PROGRAM PRG_SystemInit
VAR_OUTPUT
	bDone           : BOOL := FALSE;
END_VAR
VAR
	i               : INT;
	j				: INT;
    bAllDone        : BOOL := FALSE;
    bStartedAction  : BOOL := FALSE;
	bMoveZeroDone	: BOOL := FALSE;
    bInitComplete   : BOOL := FALSE;
	bVerticalMotorsDone		: BOOL := FALSE;   
	bLinearMotorsHomingDone	: BOOL := FALSE; 
	bValvesHomingDone 		: BOOL := FALSE;
	bLinearPumpsDone		: BOOL := FALSE;
	bPerformHoming			: BOOL := FALSE;
	
	bAllResetDone		: BOOL := FALSE;
	bEnableDone			: BOOL := FALSE;
	bResetCheck			: ARRAY[1..28] OF BOOL;
	
	aMotorsEnabled 	: ARRAY[1..3] OF BOOL;
	aValvesEnabled 	: ARRAY[1..5] OF BOOL;
	aLinearPumpsEnabled	: ARRAY[1..10] OF BOOL;
	aRotaryPumpsEnabled	: ARRAY[1..10] OF BOOL;
	
	bAllPumpsEnabled  : BOOL := FALSE;
	bAllLinearPumpsEnabled  : BOOL := FALSE;
	bAllRotaryPumpsEnabled  : BOOL := FALSE;
	bAllMotorsEnabled : BOOL := FALSE;
	bAllValvesEnabled : BOOL := FALSE;
	
	bHomeMotorDone	: ARRAY[1..3] OF BOOL;
	bHomeValveDone  : ARRAY[1..5] OF BOOL;
	bHomePumpDone	: ARRAY[1..10] OF BOOL;
	
	bM2InPosition	: BOOL;
	rPosTolerance	: REAL := 1.0;
	
	bMoveValve1Request	: BOOL := TRUE;
	bMoveValve2Request	: BOOL := TRUE;
	
	bMoveMotorsRequest	: ARRAY[1..3] OF BOOL;
	bMoveMotorDone		: ARRAY[1..3] OF BOOL;
	
	bCalibrationReset	  : BOOL := FALSE;
	bManualModeReset	  : BOOL := FALSE;
	bAutoCycleReset		  : BOOL := FALSE;
	bAllLogicResetDone	  : BOOL := FALSE;
	bInitLogicLatchesDone : BOOL := FALSE;
	
	tonResetDelay	: ton;
	tonEnableDelay	: ton;
	
	//Timeout timers for each step
	tonResetTimeOut		: ton;
	tonEnableTimeOut	: ton;
	tonHomeTimeOut		: ton;
	tonMoveAbsTimeOut	: ton;
		
	stStatus : ST_ActuatorStatus;
	
END_VAR

// ============================================================================
// PRG_SystemInit
// Handles full system initialization sequence:
//  0) Reset PRG's Manual | Calibration | AutoCycle
//  1) Reset all axes (motors, valves, pumps)
//  2) Enable all required axes
//  3) Perform homing on first startup OR move axes to zero on subsequent inits
//  4) Check completion and errors
//  5) Set bDone when initialization is complete
// ============================================================================

// ---------------------------------------------------------------------------
// 0) Basic delays between phases
// ---------------------------------------------------------------------------

// Delay before starting Reset
tonResetDelay(
    IN := NOT bAllResetDone,
    PT := T#1S
);

// Delay before starting Enable (only after Reset is fully done)
tonEnableDelay(
    IN := bAllResetDone AND NOT bEnableDone,
    PT := T#1S
);

// ---------------------------------------------------------------------------
// 0) Step 0 - Reset all logic Flags, PRGs and FBs
// ---------------------------------------------------------------------------
IF NOT bInitLogicLatchesDone THEN ACT_ResetCommandFlags(); END_IF

IF NOT bAllLogicResetDone AND bInitLogicLatchesDone THEN ACT_LogicResets(); END_IF

// ---------------------------------------------------------------------------
// 1) Step 1 - Reset all axes (motors, valves, linear and rotary pumps)
// ---------------------------------------------------------------------------
IF NOT bAllResetDone AND bAllLogicResetDone AND bInitLogicLatchesDone AND tonResetDelay.Q THEN
    ACT_ResetMotors();   // Uses bResetCheck[1..28], tonResetTimeOut, etc.
END_IF

// ---------------------------------------------------------------------------
// 2) Step 2 - Enable all axes (motors, valves, rotary pumps)
//     - Uses extra layer: checks Axis.Status.Error before/after Enable
// ---------------------------------------------------------------------------
IF bAllResetDone AND NOT bEnableDone AND tonEnableDelay.Q THEN
    ACT_EnableMotors();
END_IF

// ---------------------------------------------------------------------------
// 3) Step 3 - Decide if we need Homing or only MoveToZero
//     - First SystemInit: perform homing (bInitialHomingDone = FALSE)
//     - Next SystemInits: only move motors/valves to zero/home position
// ---------------------------------------------------------------------------

IF NOT bStartedAction AND bAllResetDone AND bEnableDone THEN
    bStartedAction := TRUE;

    // First time the machine starts: perform initial homing
    IF NOT GVL_Motion.bInitialHomingDone THEN
        bPerformHoming := TRUE;   // ACT_Homing() will be called
    ELSE
        bPerformHoming := FALSE;  // ACT_MoveToZero() will be called
    END_IF
END_IF

// ---------------------------------------------------------------------------
// 3a) Execute Homing or MoveToZero depending on bPerformHoming
// ---------------------------------------------------------------------------
IF bStartedAction THEN
    IF bPerformHoming THEN
        ACT_Homing();
    ELSE
        ACT_MoveToZero();
    END_IF
END_IF

// ---------------------------------------------------------------------------
// 4) Step 4 + 5 - Check if all motors and valves have completed their action
//     - Also checks for errors from wrapper (stStatus.bError)
//       and directly from Axis.Status.Error
// ---------------------------------------------------------------------------
IF bStartedAction AND bMoveZeroDone THEN
    bAllDone := TRUE;

    // Check motors M1..M3
    FOR i := 1 TO 3 DO
        stStatus := GVL_Motion.aMotors[i].GetStatus();

        // If any motor is not done yet
        IF NOT stStatus.bDone THEN
            bAllDone := FALSE;
        END_IF

        // If any motor returned an error (wrapper OR Axis), abort with immediate fault
        IF stStatus.bError THEN
            GVL_HMI.eMachineMode := E_MachineMode.IMEDIATE_FAULT;
            RETURN;
        END_IF
    END_FOR

    // Check valves V1..V5
    FOR i := 1 TO 5 DO
        stStatus := GVL_Motion.aValvesObj[i].GetStatus();

        // If any valve is not done yet
        IF NOT stStatus.bDone THEN
            bAllDone := FALSE;
        END_IF

        // If any valve returned an error (wrapper OR Axis), abort with immediate fault
        IF stStatus.bError THEN
            GVL_HMI.eMachineMode := E_MachineMode.IMEDIATE_FAULT;
            RETURN;
        END_IF
    END_FOR
END_IF

// ---------------------------------------------------------------------------
// 5) Step 6 - Finalization of System Init
//     - Set bDone only when Reset, Enable and Actions are all completed
// ---------------------------------------------------------------------------
IF bAllDone AND bAllResetDone AND bEnableDone AND NOT bInitComplete THEN
    bInitComplete := TRUE;
    bDone         := TRUE;

    // Mark that the initial homing has been successfully completed
    IF NOT GVL_Motion.bInitialHomingDone THEN
        GVL_Motion.bInitialHomingDone := TRUE;
    END_IF
END_IF

ACTION ACT_EnableMotors:
// ============================================================================
// Step 2: Enable all motors, valves and rotary pumps
//   - Uses aMotorsEnabled[1..3], aValvesEnabled[1..5], aRotaryPumpsEnabled[1..10]
//   - Sets bAllMotorsEnabled, bAllValvesEnabled, bAllRotaryPumpsEnabled
//   - Uses tonEnableTimeOut and GVL_Alarms.sMotionEnableTimeoutAxis
//   - Extra layer: checks wrapper error (GetStatus().bError) before enabling
// ============================================================================

IF NOT bEnableDone THEN

    // Assume all will be enabled, then AND with each device
    bAllMotorsEnabled      := TRUE;
    bAllValvesEnabled      := TRUE;
    bAllRotaryPumpsEnabled := TRUE;

    // -----------------------------
    // 2.1 Motors (M1..M3)
    // -----------------------------
    FOR i := 1 TO 3 DO
        // Read wrapper status
        stStatus := GVL_Motion.aMotors[i].GetStatus();

        // If wrapper reports error at this stage, abort System Init
        IF stStatus.bError THEN
            GVL_HMI.eMachineMode := E_MachineMode.IMEDIATE_FAULT;
            RETURN;
        END_IF

        // If axis is disabled, request Enable through wrapper
        // (If your wrapper has a specific bEnabled flag, you can check it here.
        // Otherwise, just call Enable() and rely on the wrapper to handle it.)
        aMotorsEnabled[i] := GVL_Motion.aMotors[i].Enable();

        bAllMotorsEnabled := bAllMotorsEnabled AND aMotorsEnabled[i];
    END_FOR

    // -----------------------------
    // 2.2 Valves (V1..V5)
    // -----------------------------
    FOR i := 1 TO 5 DO
        stStatus := GVL_Motion.aValvesObj[i].GetStatus();

        IF stStatus.bError THEN
            GVL_HMI.eMachineMode := E_MachineMode.IMEDIATE_FAULT;
            RETURN;
        END_IF

        aValvesEnabled[i] := GVL_Motion.aValvesObj[i].Enable();

        bAllValvesEnabled := bAllValvesEnabled AND aValvesEnabled[i];
    END_FOR

    // -----------------------------
    // 2.3 Rotary pumps (RP1..RP10)
// -----------------------------
    FOR i := 1 TO 10 DO
        stStatus := GVL_Motion.aPumpsRotary[i].GetStatus();

        IF stStatus.bError THEN
            GVL_HMI.eMachineMode := E_MachineMode.IMEDIATE_FAULT;
            RETURN;
        END_IF

        aRotaryPumpsEnabled[i] := GVL_Motion.aPumpsRotary[i].Enable();

        bAllRotaryPumpsEnabled := bAllRotaryPumpsEnabled AND aRotaryPumpsEnabled[i];
    END_FOR

    // -----------------------------
    // 2.4 Enable timeout monitoring and alarm
    // -----------------------------
    tonEnableTimeOut(IN := TRUE, PT := T#10S);

    IF tonEnableTimeOut.Q AND NOT (bAllMotorsEnabled AND bAllValvesEnabled AND bAllRotaryPumpsEnabled) THEN
        // Build string with axes that were NOT enabled within timeout

        // Motors M1..M3
        FOR i := 1 TO 3 DO
            IF NOT aMotorsEnabled[i] THEN
                IF GVL_Alarms.sMotionEnableTimeoutAxis <> '' THEN
                    GVL_Alarms.sMotionEnableTimeoutAxis :=
                        CONCAT(GVL_Alarms.sMotionEnableTimeoutAxis, ', ');
                END_IF
                GVL_Alarms.sMotionEnableTimeoutAxis :=
                    CONCAT(GVL_Alarms.sMotionEnableTimeoutAxis,
                           GVL_Constant.sMotionText[i]);
            END_IF
        END_FOR

        // Valves V1..V5
        FOR i := 1 TO 5 DO
            IF NOT aValvesEnabled[i] THEN
                IF GVL_Alarms.sMotionEnableTimeoutAxis <> '' THEN
                    GVL_Alarms.sMotionEnableTimeoutAxis :=
                        CONCAT(GVL_Alarms.sMotionEnableTimeoutAxis, ', ');
                END_IF
                GVL_Alarms.sMotionEnableTimeoutAxis :=
                    CONCAT(GVL_Alarms.sMotionEnableTimeoutAxis,
                           GVL_Constant.sMotionText[i + 3]);
            END_IF
        END_FOR

        // Rotary pumps RP1..RP10
        FOR i := 1 TO 10 DO
            IF NOT aRotaryPumpsEnabled[i] THEN
                IF GVL_Alarms.sMotionEnableTimeoutAxis <> '' THEN
                    GVL_Alarms.sMotionEnableTimeoutAxis :=
                        CONCAT(GVL_Alarms.sMotionEnableTimeoutAxis, ', ');
                END_IF
                GVL_Alarms.sMotionEnableTimeoutAxis :=
                    CONCAT(GVL_Alarms.sMotionEnableTimeoutAxis,
                           GVL_Constant.sMotionText[i + 18]);
            END_IF
        END_FOR

        GVL_Alarms.bMotionEnableTimeout := TRUE;
        // Strong robustness: abort System Init on enable timeout
        GVL_HMI.eMachineMode := E_MachineMode.IMEDIATE_FAULT;
        RETURN;
    END_IF

    // -----------------------------
    // 2.5 Step completion
    // -----------------------------
    IF bAllMotorsEnabled AND bAllValvesEnabled AND bAllRotaryPumpsEnabled THEN
        bEnableDone := TRUE;
        tonEnableTimeOut(IN := FALSE);
    END_IF

ELSE
    // Already done, ensure timer is off
    tonEnableTimeOut(IN := FALSE);
END_IF
END_ACTION

ACTION ACT_Homing:
// ============================================================================
// Step 3 (part 1): Initial homing sequence
//   - Only used when GVL_Motion.bInitialHomingDone = FALSE
//   - Homes vertical motors, then horizontal motor
//   - Moves valves to home position (position 5) when positions are recovered
//   - Monitors homing timeout and raises alarm
// ============================================================================

IF bPerformHoming THEN

    // -----------------------------
    // 3.1 Vertical motors homing (M1, M2)
    // -----------------------------
    IF NOT bHomeMotorDone[1] THEN
        bHomeMotorDone[1] := GVL_Motion.aMotors[1].Home(
            pHomeSensor := ADR(GVL_IO.gDigInputs.bStageCollection_Home),
            rVelocity   := GVL_Motion.M1Motor.rHomeVel,
            rAcc        := GVL_Motion.M1Motor.rHomeAcc,
            rDec        := GVL_Motion.M1Motor.rHomeDec
        );
    END_IF

    IF NOT bHomeMotorDone[2] THEN
        bHomeMotorDone[2] := GVL_Motion.aMotors[2].Home(
            pHomeSensor := ADR(GVL_IO.gDigInputs.bSampleRecovery_Vertical_Home),
            rVelocity   := GVL_Motion.M2Motor.rHomeVel,
            rAcc        := GVL_Motion.M2Motor.rHomeAcc,
            rDec        := GVL_Motion.M2Motor.rHomeDec
        );
    END_IF

    // Check if vertical motors homing is done
    IF bHomeMotorDone[1] AND bHomeMotorDone[2] THEN
        bVerticalMotorsDone := TRUE;
    END_IF

    // -----------------------------
    // 3.2 Horizontal motor homing (M3), only after verticals are done
    // -----------------------------
    IF bVerticalMotorsDone AND NOT bHomeMotorDone[3] THEN
        bHomeMotorDone[3] := GVL_Motion.aMotors[3].Home(
            pHomeSensor := ADR(GVL_IO.gDigInputs.bSampleRecovery_Horizontal_Home),
            rVelocity   := GVL_Motion.M3Motor.rHomeVel,
            rAcc        := GVL_Motion.M3Motor.rHomeAcc,
            rDec        := GVL_Motion.M3Motor.rHomeDec
        );
    END_IF

    // Check if all linear motors are homed
    IF bHomeMotorDone[1] AND bHomeMotorDone[2] AND bHomeMotorDone[3] THEN
        bLinearMotorsHomingDone := TRUE;
    END_IF

    // -----------------------------
    // 3.3 Valves homing (move to position 5) if position is recovered
    // -----------------------------
    IF GVL_Motion.bValvesPositionRecovered THEN
        // Move all valves to position 5 (home position)
        IF NOT bHomeValveDone[1] THEN
            bHomeValveDone[1] := GVL_Motion.aValvesObj[1].MoveValve(
                iPosition := 5,
                rVelocity := GVL_Motion.aValves[1].rHomeVel,
                rAcc      := GVL_Motion.aValves[1].rHomeAcc,
                rDec      := GVL_Motion.aValves[1].rHomeDec
            );
        END_IF

        IF NOT bHomeValveDone[2] THEN
            bHomeValveDone[2] := GVL_Motion.aValvesObj[2].MoveValve(
                iPosition := 5,
                rVelocity := GVL_Motion.aValves[2].rHomeVel,
                rAcc      := GVL_Motion.aValves[2].rHomeAcc,
                rDec      := GVL_Motion.aValves[2].rHomeDec
            );
        END_IF

        IF NOT bHomeValveDone[3] THEN
            bHomeValveDone[3] := GVL_Motion.aValvesObj[3].MoveValve(
                iPosition := 5,
                rVelocity := GVL_Motion.aValves[3].rHomeVel,
                rAcc      := GVL_Motion.aValves[3].rHomeAcc,
                rDec      := GVL_Motion.aValves[3].rHomeDec
            );
        END_IF

        IF NOT bHomeValveDone[4] THEN
            bHomeValveDone[4] := GVL_Motion.aValvesObj[4].MoveValve(
                iPosition := 5,
                rVelocity := GVL_Motion.aValves[4].rHomeVel,
                rAcc      := GVL_Motion.aValves[4].rHomeAcc,
                rDec      := GVL_Motion.aValves[4].rHomeDec
            );
        END_IF

        IF NOT bHomeValveDone[5] THEN
            bHomeValveDone[5] := GVL_Motion.aValvesObj[5].MoveValve(
                iPosition := 5,
                rVelocity := GVL_Motion.aValves[5].rHomeVel,
                rAcc      := GVL_Motion.aValves[5].rHomeAcc,
                rDec      := GVL_Motion.aValves[5].rHomeDec
            );
        END_IF
    END_IF

    // Check if all valves homing are done
    bValvesHomingDone :=
        bHomeValveDone[1] AND bHomeValveDone[2] AND bHomeValveDone[3] AND
        bHomeValveDone[4] AND bHomeValveDone[5];

	// If all motors and valves completed their homing, finalize
	IF bLinearMotorsHomingDone AND bValvesHomingDone THEN 
		bMoveZeroDone := TRUE;
	END_IF	
	
    // -----------------------------
    // 3.4 Homing timeout monitoring and alarm
    // -----------------------------
    tonHomeTimeOut(
        IN := NOT (bLinearMotorsHomingDone AND bValvesHomingDone),
        PT := T#40S
    );

    IF tonHomeTimeOut.Q AND NOT (bLinearMotorsHomingDone AND bValvesHomingDone) THEN
        // Build string with axes that were NOT homed in time

        // Motors M1..M3
        FOR j := 1 TO 3 DO
            IF NOT bHomeMotorDone[j] THEN
                IF GVL_Alarms.sMotionHomeTimeoutAxis <> '' THEN
                    GVL_Alarms.sMotionHomeTimeoutAxis :=
                        CONCAT(GVL_Alarms.sMotionHomeTimeoutAxis, ', ');
                END_IF
                GVL_Alarms.sMotionHomeTimeoutAxis :=
                    CONCAT(GVL_Alarms.sMotionHomeTimeoutAxis,
                           GVL_Constant.sMotionText[j]);
            END_IF
        END_FOR

        // Valves V1..V5
        FOR j := 1 TO 5 DO
            IF NOT bHomeValveDone[j] THEN
                IF GVL_Alarms.sMotionHomeTimeoutAxis <> '' THEN
                    GVL_Alarms.sMotionHomeTimeoutAxis :=
                        CONCAT(GVL_Alarms.sMotionHomeTimeoutAxis, ', ');
                END_IF
                GVL_Alarms.sMotionHomeTimeoutAxis :=
                    CONCAT(GVL_Alarms.sMotionHomeTimeoutAxis,
                           GVL_Constant.sMotionText[j + 3]);
            END_IF
        END_FOR

        GVL_Alarms.bMotionHomeTimeout := TRUE;
        GVL_HMI.eMachineMode          := E_MachineMode.IMEDIATE_FAULT;
    END_IF

END_IF
END_ACTION

ACTION ACT_LogicResets:
IF NOT bAllLogicResetDone THEN
	
	bCalibrationReset	:= PRG_Calibration.Reset();
	bManualModeReset	:= PRG_ManualControl.Reset();
	bAutoCycleReset		:= PRG_AutoCycle.Reset();
	
	IF bCalibrationReset AND bManualModeReset AND bAutoCycleReset THEN
		bAllLogicResetDone 	:= TRUE;
	END_IF
	
END_IF
END_ACTION

ACTION ACT_MoveToZero:
// ============================================================================
// Step 3 (part 2): Move motors and valves to zero / default positions
//   - Used when GVL_Motion.bInitialHomingDone = TRUE
//   - Moves:
//       - M1, M2, M3 -> position 0.0
//       - Valves V1..V5 -> position 5
//   - Uses bMoveMotorDone[1..3] and bHomeValveDone[1..5]
//   - Monitors move absolute timeout and raises alarm
// ============================================================================

IF NOT bPerformHoming THEN

    // -----------------------------
    // 3.5 Move linear motors to 0.0
    // -----------------------------
    // You can adjust these velocity/acc/dec parameters as needed
    IF NOT bMoveMotorDone[1] THEN
        bMoveMotorDone[1] := GVL_Motion.aMotors[1].MoveAbsolute(
            rPosition := GVL_Settings.stMachineParam.aM1Position[1],
            rVelocity := GVL_Settings.stMachineParam.rM1Velocity,
            rAcc      := GVL_Settings.stMachineParam.rM1Accleration,
            rDec      := GVL_Settings.stMachineParam.rM1Deceleration
        );
    END_IF

    IF NOT bMoveMotorDone[2] THEN
        bMoveMotorDone[2] := GVL_Motion.aMotors[2].MoveAbsolute(
            rPosition := GVL_Settings.stMachineParam.aM2Position[1],
            rVelocity := GVL_Settings.stMachineParam.rM2Velocity,
            rAcc      := GVL_Settings.stMachineParam.rM2Accleration,
            rDec      := GVL_Settings.stMachineParam.rM2Deceleration
        );
    END_IF
	
	// Track real M2 Position before start moving M3 
	bM2InPosition := ABS(GVL_Motion.M2Motor.rActualPos - GVL_Settings.stMachineParam.aM2Position[1]) < rPosTolerance;
	
    IF bMoveMotorDone[2] AND bM2InPosition AND NOT bMoveMotorDone[3] THEN
        bMoveMotorDone[3] := GVL_Motion.aMotors[3].MoveAbsolute(
            rPosition := GVL_Settings.stMachineParam.aM3Position[1],
            rVelocity := GVL_Settings.stMachineParam.rM3Velocity,
            rAcc      := GVL_Settings.stMachineParam.rM3Accleration,
            rDec      := GVL_Settings.stMachineParam.rM3Deceleration
        );
    END_IF

    // Linear motors move done flag
    bLinearMotorsHomingDone :=
        bMoveMotorDone[1] AND bMoveMotorDone[2] AND bMoveMotorDone[3];

    // -----------------------------
    // 3.6 Move valves to position 5 (default/home position)
// -----------------------------
    IF NOT bHomeValveDone[1] THEN
        bHomeValveDone[1] := GVL_Motion.aValvesObj[1].MoveValve(
            iPosition := 5,
            rVelocity := GVL_Motion.aValves[1].rHomeVel,
            rAcc      := GVL_Motion.aValves[1].rHomeAcc,
            rDec      := GVL_Motion.aValves[1].rHomeDec
        );
    END_IF

    IF NOT bHomeValveDone[2] THEN
        bHomeValveDone[2] := GVL_Motion.aValvesObj[2].MoveValve(
            iPosition := 5,
            rVelocity := GVL_Motion.aValves[2].rHomeVel,
            rAcc      := GVL_Motion.aValves[2].rHomeAcc,
            rDec      := GVL_Motion.aValves[2].rHomeDec
        );
    END_IF

    IF NOT bHomeValveDone[3] THEN
        bHomeValveDone[3] := GVL_Motion.aValvesObj[3].MoveValve(
            iPosition := 5,
            rVelocity := GVL_Motion.aValves[3].rHomeVel,
            rAcc      := GVL_Motion.aValves[3].rHomeAcc,
            rDec      := GVL_Motion.aValves[3].rHomeDec
        );
    END_IF

    IF NOT bHomeValveDone[4] THEN
        bHomeValveDone[4] := GVL_Motion.aValvesObj[4].MoveValve(
            iPosition := 5,
            rVelocity := GVL_Motion.aValves[4].rHomeVel,
            rAcc      := GVL_Motion.aValves[4].rHomeAcc,
            rDec      := GVL_Motion.aValves[4].rHomeDec
        );
    END_IF

    IF NOT bHomeValveDone[5] THEN
        bHomeValveDone[5] := GVL_Motion.aValvesObj[5].MoveValve(
            iPosition := 5,
            rVelocity := GVL_Motion.aValves[5].rHomeVel,
            rAcc      := GVL_Motion.aValves[5].rHomeAcc,
            rDec      := GVL_Motion.aValves[5].rHomeDec
        );
    END_IF

    // Valves move done flag
    bValvesHomingDone :=
        bHomeValveDone[1] AND bHomeValveDone[2] AND
        bHomeValveDone[3] AND bHomeValveDone[4] AND bHomeValveDone[5];
	
	// If all motors and valves completed their homing, finalize
	IF bLinearMotorsHomingDone AND bValvesHomingDone THEN 
		bMoveZeroDone := TRUE;
	END_IF
	
    // -----------------------------
    // 3.7 MoveAbs timeout monitoring and alarm
    //    (Note: here we correctly use bMoveMotorDone instead of bHomeMotorDone)
// -----------------------------
    tonMoveAbsTimeOut(
        IN := NOT (bLinearMotorsHomingDone AND bValvesHomingDone),
        PT := T#40S
    );

    IF tonMoveAbsTimeOut.Q AND NOT (bLinearMotorsHomingDone AND bValvesHomingDone) THEN
        // Build string with axes that did NOT complete MoveAbsolute in time

        // Motors M1..M3
        FOR j := 1 TO 3 DO
            IF NOT bMoveMotorDone[j] THEN
                IF GVL_Alarms.sMotionMoveAbsTimeoutAxis <> '' THEN
                    GVL_Alarms.sMotionMoveAbsTimeoutAxis :=
                        CONCAT(GVL_Alarms.sMotionMoveAbsTimeoutAxis, ', ');
                END_IF
                GVL_Alarms.sMotionMoveAbsTimeoutAxis :=
                    CONCAT(GVL_Alarms.sMotionMoveAbsTimeoutAxis,
                           GVL_Constant.sMotionText[j]);
            END_IF
        END_FOR

        // Valves V1..V5
        FOR j := 1 TO 5 DO
            IF NOT bHomeValveDone[j] THEN
                IF GVL_Alarms.sMotionMoveAbsTimeoutAxis <> '' THEN
                    GVL_Alarms.sMotionMoveAbsTimeoutAxis :=
                        CONCAT(GVL_Alarms.sMotionMoveAbsTimeoutAxis, ', ');
                END_IF
                GVL_Alarms.sMotionMoveAbsTimeoutAxis :=
                    CONCAT(GVL_Alarms.sMotionMoveAbsTimeoutAxis,
                           GVL_Constant.sMotionText[j + 3]);
            END_IF
        END_FOR

        GVL_Alarms.bMotionMoveAbsTimeout := TRUE;
        GVL_HMI.eMachineMode             := E_MachineMode.IMEDIATE_FAULT;
    END_IF

END_IF
END_ACTION

ACTION ACT_ResetCommandFlags:
(*
    Action: ACT_ResetCommandFlags
    Purpose:
        Clear all HMI command flags and internal latched commands that might remain TRUE
        after an abnormal interruption (STOP/Abort), preventing unintended auto-start
        when re-entering a mode.

    Where to call:
        - PRG_StoppedState (first scan / when entering STOPPED)
        - PRG_SystemInit (first scan / at init start)

    Notes:
        - This action is safe to call repeatedly (idempotent).
        - Adjust array bounds if your project differs.
*)

// ============================================================
// 1) Calibration - HMI triggers (buttons / commands)
// ============================================================
GVL_HMI.bStartCalibrationBt        := FALSE;

GVL_HMI.bCalLeakTestButton         := FALSE;
GVL_HMI.bCalPressureUpSystemBt     := FALSE;
GVL_HMI.bCalHoldSysPressureBt      := FALSE;
GVL_HMI.bCalStopLeakTestBt         := FALSE;

GVL_HMI.bCalLinearPumpsEnableBt    := FALSE;
GVL_HMI.bCalLinearPumpsHomeBt      := FALSE;
GVL_HMI.bCalLinearPumpsMoveBt      := FALSE;
GVL_HMI.bCalLinearPumpsStopBt      := FALSE;
GVL_HMI.bCalLinearPumpsDirty       := FALSE;

GVL_HMI.bCalMoveValves             := FALSE;
GVL_HMI.bCalMoveM1Motor            := FALSE;

// Scale / CalBox popups / acknowledge flags
GVL_HMI.bScaleNeedsAtention        := FALSE;
GVL_HMI.bScaleFixed                := FALSE;
GVL_HMI.bCalBoxNeedsAttention      := FALSE;
GVL_HMI.bCalBoxFixed               := FALSE;


// ============================================================
// 2) Calibration - internal latches (must be cleared on STOP/Init)
// ============================================================
GVL_Calibration.bStartCalibration      := FALSE;
GVL_Calibration.bAbortCalibration      := FALSE;
GVL_Calibration.bStartCreationCalJson  := FALSE;


// ============================================================
// 3) Manual Mode - motors / valves / pumps command arrays
// ============================================================

// Manual motors (adjust bounds if needed)
FOR i := 1 TO 3 DO
    GVL_HMI.aManualMotorsCmd[i].bRun  := FALSE;
    GVL_HMI.aManualMotorsCmd[i].bStop := FALSE;
END_FOR

// Manual valves
FOR i := 1 TO 5 DO
    GVL_HMI.aManualValvesCmd[i].bMove := FALSE;
    GVL_HMI.aManualValvesCmd[i].bStop := FALSE;
END_FOR

// Global pump buttons
GVL_HMI.bRunPumpsBySpeedBt  := FALSE;
GVL_HMI.bRunPumpsByVolumeBt := FALSE;

// Per-pump commands
FOR i := 1 TO 10 DO
    GVL_HMI.aManualPumpsCmd[i].bRunBySpeed  := FALSE;
    GVL_HMI.aManualPumpsCmd[i].bRunByVolume := FALSE;
    GVL_HMI.aManualPumpsCmd[i].bStop        := FALSE;
    GVL_HMI.aManualPumpsCmd[i].bActive      := FALSE;
END_FOR


// ============================================================
// 4) AutoCycle - popup/start/hold commands
// ============================================================
GVL_HMI.bShowAutoCyclePopup     	:= FALSE;
GVL_HMI.bStartAutoCycleButton   	:= FALSE;
GVL_HMI.bSystemReady_ReqAutoCycle 	:= FALSE;

GVL_HMI.bAutoCycleHoldReq       	:= FALSE;
GVL_HMI.bAutoCycleHoldActive    	:= FALSE;
GVL_HMI.bAutoCycleHoldPopup     	:= FALSE;
GVL_HMI.bAutoCycleContinueCmd   	:= FALSE;
GVL_HMI.bAutoCycleCancelCmd     	:= FALSE;


// ============================================================
// 5) Finishing
// ============================================================
bInitLogicLatchesDone := TRUE;
END_ACTION

ACTION ACT_ResetMotors:
// ============================================================================
// Step 1: Reset all motors, valves, linear and rotary pumps
// Uses array bResetCheck[1..28] to track each device:
//   1..3   -> Motors      (M1..M3)
//   4..8   -> Valves      (V1..V5)
//   9..18  -> Linear pumps  (LP1..LP10)
//   19..28 -> Rotary pumps  (RP1..RP10)
// ============================================================================

IF NOT bAllResetDone THEN

    // -----------------------------
    // 1.1 Motors (M1..M3)
    // -----------------------------
    IF NOT bResetCheck[1] THEN
        bResetCheck[1] := GVL_Motion.aMotors[1].Reset();
    END_IF

    IF NOT bResetCheck[2] THEN
        bResetCheck[2] := GVL_Motion.aMotors[2].Reset();
    END_IF

    IF NOT bResetCheck[3] THEN
        bResetCheck[3] := GVL_Motion.aMotors[3].Reset();
    END_IF

    // -----------------------------
    // 1.2 Valves (V1..V5)
    // -----------------------------
    IF NOT bResetCheck[4] THEN
        bResetCheck[4] := GVL_Motion.aValvesObj[1].Reset();
    END_IF

    IF NOT bResetCheck[5] THEN
        bResetCheck[5] := GVL_Motion.aValvesObj[2].Reset();
    END_IF

    IF NOT bResetCheck[6] THEN
        bResetCheck[6] := GVL_Motion.aValvesObj[3].Reset();
    END_IF

    IF NOT bResetCheck[7] THEN
        bResetCheck[7] := GVL_Motion.aValvesObj[4].Reset();
    END_IF

    IF NOT bResetCheck[8] THEN
        bResetCheck[8] := GVL_Motion.aValvesObj[5].Reset();
    END_IF

    // -----------------------------
    // 1.3 Linear pumps (LP1..LP10)
    // -----------------------------
    IF NOT bResetCheck[9] THEN
        bResetCheck[9] := GVL_Motion.aPumpsLinear[1].Reset();
    END_IF
    IF NOT bResetCheck[10] THEN
        bResetCheck[10] := GVL_Motion.aPumpsLinear[2].Reset();
    END_IF
    IF NOT bResetCheck[11] THEN
        bResetCheck[11] := GVL_Motion.aPumpsLinear[3].Reset();
    END_IF
    IF NOT bResetCheck[12] THEN
        bResetCheck[12] := GVL_Motion.aPumpsLinear[4].Reset();
    END_IF
    IF NOT bResetCheck[13] THEN
        bResetCheck[13] := GVL_Motion.aPumpsLinear[5].Reset();
    END_IF
    IF NOT bResetCheck[14] THEN
        bResetCheck[14] := GVL_Motion.aPumpsLinear[6].Reset();
    END_IF
    IF NOT bResetCheck[15] THEN
        bResetCheck[15] := GVL_Motion.aPumpsLinear[7].Reset();
    END_IF
    IF NOT bResetCheck[16] THEN
        bResetCheck[16] := GVL_Motion.aPumpsLinear[8].Reset();
    END_IF
    IF NOT bResetCheck[17] THEN
        bResetCheck[17] := GVL_Motion.aPumpsLinear[9].Reset();
    END_IF
    IF NOT bResetCheck[18] THEN
        bResetCheck[18] := GVL_Motion.aPumpsLinear[10].Reset();
    END_IF

    // -----------------------------
    // 1.4 Rotary pumps (RP1..RP10)
    // -----------------------------
    IF NOT bResetCheck[19] THEN
        bResetCheck[19] := GVL_Motion.aPumpsRotary[1].Reset();
    END_IF
    IF NOT bResetCheck[20] THEN
        bResetCheck[20] := GVL_Motion.aPumpsRotary[2].Reset();
    END_IF
    IF NOT bResetCheck[21] THEN
        bResetCheck[21] := GVL_Motion.aPumpsRotary[3].Reset();
    END_IF
    IF NOT bResetCheck[22] THEN
        bResetCheck[22] := GVL_Motion.aPumpsRotary[4].Reset();
    END_IF
    IF NOT bResetCheck[23] THEN
        bResetCheck[23] := GVL_Motion.aPumpsRotary[5].Reset();
    END_IF
    IF NOT bResetCheck[24] THEN
        bResetCheck[24] := GVL_Motion.aPumpsRotary[6].Reset();
    END_IF
    IF NOT bResetCheck[25] THEN
        bResetCheck[25] := GVL_Motion.aPumpsRotary[7].Reset();
    END_IF
    IF NOT bResetCheck[26] THEN
        bResetCheck[26] := GVL_Motion.aPumpsRotary[8].Reset();
    END_IF
    IF NOT bResetCheck[27] THEN
        bResetCheck[27] := GVL_Motion.aPumpsRotary[9].Reset();
    END_IF
    IF NOT bResetCheck[28] THEN
        bResetCheck[28] := GVL_Motion.aPumpsRotary[10].Reset();
    END_IF

    // -----------------------------------------------------------------------
    // 1.5 Check if all resets are done
    // -----------------------------------------------------------------------
    IF bResetCheck[1] AND bResetCheck[2] AND bResetCheck[3] AND
       bResetCheck[4] AND bResetCheck[5] AND bResetCheck[6] AND
       bResetCheck[7] AND bResetCheck[8] AND
       bResetCheck[9] AND bResetCheck[10] AND bResetCheck[11] AND
       bResetCheck[12] AND bResetCheck[13] AND bResetCheck[14] AND
       bResetCheck[15] AND bResetCheck[16] AND bResetCheck[17] AND
       bResetCheck[18] AND
       bResetCheck[19] AND bResetCheck[20] AND bResetCheck[21] AND
       bResetCheck[22] AND bResetCheck[23] AND bResetCheck[24] AND
       bResetCheck[25] AND bResetCheck[26] AND bResetCheck[27] AND
       bResetCheck[28] THEN
        bAllResetDone := TRUE;
    ELSE
        bAllResetDone := FALSE;
    END_IF

    // -----------------------------------------------------------------------
    // 1.6 Reset timeout monitoring and alarm trigger
    // -----------------------------------------------------------------------
    tonResetTimeOut(IN := TRUE, PT := T#10S);

    IF tonResetTimeOut.Q THEN
        // Build string with axes that were NOT reset within timeout
        FOR j := 1 TO 28 DO
            IF NOT bResetCheck[j] THEN
                IF GVL_Alarms.sMotionResetTimeoutAxis <> '' THEN
                    GVL_Alarms.sMotionResetTimeoutAxis :=
                        CONCAT(GVL_Alarms.sMotionResetTimeoutAxis, ', ');
                END_IF
                GVL_Alarms.sMotionResetTimeoutAxis :=
                    CONCAT(GVL_Alarms.sMotionResetTimeoutAxis,
                           GVL_Constant.sMotionText[j]);
            END_IF
        END_FOR

        GVL_Alarms.bMotionResetTimeout := TRUE;
        // Optional: you could also force IMEDIATE_FAULT here if desired
    END_IF

ELSE
    // Reset already completed, ensure timeout timer is off
    tonResetTimeOut(IN := FALSE);
END_IF
END_ACTION

METHOD Reset : BOOL
VAR_INPUT	
END_VAR
VAR
	i : INT;
END_VAR
// ============================================================================
// PRG_SystemInit.Reset()
// ---------------------------------------------------------------------------
// This method clears all internal flags, arrays and timers used by
// PRG_SystemInit so that a new initialization sequence can start from a
// clean state.
//
// Return:
//   TRUE  - Always returns TRUE after the internal context is fully reset.
//           (The actual System Init progress is controlled by bAllResetDone,
//            bEnableDone, bAllDone, etc. in the main body.)
//
// Typical usage (in PRG_MasterControl):
//   - When entering E_MachineMode.SYSTEM_INITIALIZING,
//     call PRG_SystemInit.Reset() once to clear the context.
// ============================================================================

Reset := FALSE; // Default return

// ---------------------------------------------------------------------------
// 1) Global step control flags
// ---------------------------------------------------------------------------
bAllResetDone           := FALSE;
bEnableDone             := FALSE;
bStartedAction          := FALSE;
bPerformHoming          := FALSE;
bInitComplete           := FALSE;
bAllDone                := FALSE;
bMoveZeroDone 			:= FALSE;
bM2InPosition			:= FALSE;
bDone                   := FALSE;   

bVerticalMotorsDone     := FALSE;
bLinearMotorsHomingDone := FALSE;
bValvesHomingDone       := FALSE;

bCalibrationReset 		:= FALSE;
bManualModeReset 		:= FALSE;
bAutoCycleReset	 		:= FALSE;
bAllLogicResetDone 		:= FALSE;
bInitLogicLatchesDone	:= FALSE;

// ---------------------------------------------------------------------------
// 2) Per-device reset tracking array (1..28)
//    1..3   -> Motors       (M1..M3)
//    4..8   -> Valves       (V1..V5)
//    9..18  -> Linear pumps (LP1..LP10)
//    19..28 -> Rotary pumps (RP1..RP10)
// ---------------------------------------------------------------------------
FOR i := 1 TO 28 DO
    bResetCheck[i] := FALSE;
END_FOR

// ---------------------------------------------------------------------------
// 3) Enable state arrays
//    Motors:        aMotorsEnabled[1..3]
//    Valves:        aValvesEnabled[1..5]
//    Rotary pumps:  aRotaryPumpsEnabled[1..10]
// ---------------------------------------------------------------------------
FOR i := 1 TO 3 DO
    aMotorsEnabled[i] := FALSE;
END_FOR

FOR i := 1 TO 5 DO
    aValvesEnabled[i] := FALSE;
END_FOR

FOR i := 1 TO 10 DO
    aRotaryPumpsEnabled[i] := FALSE;
END_FOR

bAllMotorsEnabled      := FALSE;
bAllValvesEnabled      := FALSE;
bAllRotaryPumpsEnabled := FALSE;

// ---------------------------------------------------------------------------
// 4) Homing / MoveToZero flags
//    - bHomeMotorDone[1..3] : homing done flags for M1..M3
//    - bMoveMotorDone[1..3] : move-to-zero done flags for M1..M3
//    - bHomeValveDone[1..5] : homing/move done flags for V1..V5
// ---------------------------------------------------------------------------
FOR i := 1 TO 3 DO
    bHomeMotorDone[i] := FALSE;
    bMoveMotorDone[i] := FALSE;
END_FOR

FOR i := 1 TO 5 DO
    bHomeValveDone[i] := FALSE;
END_FOR

// ---------------------------------------------------------------------------
// 5) Timers used in System Init
// ---------------------------------------------------------------------------

// Phase delays
tonResetDelay(IN := FALSE);
tonEnableDelay(IN := FALSE);

// Timeouts
tonResetTimeOut(IN := FALSE);
tonEnableTimeOut(IN := FALSE);
tonHomeTimeOut(IN := FALSE);
tonMoveAbsTimeOut(IN := FALSE);

// ---------------------------------------------------------------------------
// 6) Alarm strings and flags used by System Init
// ---------------------------------------------------------------------------

// Reset timeout
GVL_Alarms.sMotionResetTimeoutAxis := '';
GVL_Alarms.bMotionResetTimeout     := FALSE;

// Enable timeout
GVL_Alarms.sMotionEnableTimeoutAxis := '';
GVL_Alarms.bMotionEnableTimeout     := FALSE;

// Homing timeout
GVL_Alarms.sMotionHomeTimeoutAxis := '';
GVL_Alarms.bMotionHomeTimeout     := FALSE;

// Move Absolute timeout
GVL_Alarms.sMotionMoveAbsTimeoutAxis := '';
GVL_Alarms.bMotionMoveAbsTimeout     := FALSE;

// ---------------------------------------------------------------------------
// 7) Finalize
// ---------------------------------------------------------------------------
Reset := TRUE;
END_METHOD

END_PROGRAM

(* stored: Version 1.1.0.1, ProductVersion 3.1.4024.15
   POU PRG_SystemInit: Id {de7516f5-b372-4654-9a26-44141ec2f79b}, SpecialFunc None
   Action ACT_EnableMotors: Id {d9d400bf-ab34-4cad-bf34-4bdfcfba06a2}
   Action ACT_Homing: Id {5b9a9a21-bf87-474a-922f-0cf75f21e89d}
   Action ACT_LogicResets: Id {93d90275-251c-4388-98d6-ad6cf2cf0425}
   Action ACT_MoveToZero: Id {87199ab2-9943-4068-ba24-dfc8b517e9be}
   Action ACT_ResetCommandFlags: Id {b3a2d6e7-e76c-4702-9ecb-55034b8fa2f1}
   Action ACT_ResetMotors: Id {827879fc-000a-4b08-b7c6-194c29783c28}
   Method Reset: Id {9d292ea2-dd87-459a-a476-a8e8f5acf2de} *)
